// Converts a BYTE to an ascii character
FUNCTION F_ByteToChar : T_Char
VAR_INPUT
	nByte : BYTE;
END_VAR

F_ByteToChar[0] := nByte;

END_FUNCTION

(* stored: Version 1.1.0.1, ProductVersion 3.1.4024.4
   POU F_ByteToChar: Id {cc9ba165-219c-491b-8479-7738e7a1894d}, SpecialFunc None *)
